FUNCTION_BLOCK FB_Floor
VAR_INPUT
END_VAR
VAR_OUTPUT
END_VAR
VAR
	_aRooms		: ARRAY [1..20] OF FB_Room;
END_VAR

METHOD CalcPowerConsumption : UDINT
VAR
	nRoom		: INT;
END_VAR
FOR nRoom := 1 TO 20 DO	
	CalcPowerConsumption := CalcPowerConsumption + refRooms[nRoom].CalcPowerConsumption();
END_FOR
END_METHOD

PROPERTY refRooms : REFERENCE TO ARRAY [1..20] OF FB_Room
GET
refRooms REF= THIS^._aRooms;
END_GET
END_PROPERTY

END_FUNCTION_BLOCK

(* stored: Version 1.1.0.1, ProductVersion 3.1.4024.12
   POU FB_Floor: Id {5283b3f7-f5ae-4c20-97af-7f8c264ab6b4}, SpecialFunc None
   Method CalcPowerConsumption: Id {265595fe-7771-4b20-827c-bb279464e589}
   Property refRooms: Id {7dc87f9e-c7b7-4487-90eb-e7e4b8e931b2}
   Get Get: Id {83b4a601-f8a9-4884-a468-a6c1a54f1f9d} *)
